Staubli VAL3: dataStreamer.pgx

public program dataStreamer()
begin
  while (bSendData)
    // fetch current joint positions
    jCurrPose=herej()
    // encode and send ROS simple_message ID 10: joint state
    call encodeJState()
    call sendJState()

    // fetch robot status
    call fetchStatus()
    // encode and send ROS simple_message ID 13: robot status
    call encodeStatus()
    call sendStatus()

    // sequence task
    delay(0)
  endWhile
end
